// TIA Portal V16 export
// export: Created 2021-09-08T12:46:16.4114193Z, ExportSetting WithDefaults, DisplayName Totally Integrated Automation Portal, DisplayVersion V16 Update 3, DisplayName TIA Portal Version Control Interface, DisplayVersion V16 Update 2, DisplayName TIA Portal Openness, DisplayVersion V16 Update 3, DisplayName TIA Portal Teamcenter Gateway, DisplayVersion V16, DisplayName STEP 7 Professional, DisplayVersion V16 Update 3, DisplayName STEP 7 Safety, DisplayVersion V16, DisplayName WinCC Advanced, DisplayVersion V16 Update 3
TYPE "UF_PARAMETRS"
// stored: IsFailsafeCompliant false
   STRUCT
      Sf : Real;   // Filtration square m2
      flux : Real;
      dP : Real;   // Delta preassure
      Rec : Real;   // Recovery
      Ts : UInt;   // Step time
      Tf : UDInt;   // Filtration time
   END_STRUCT;
END_TYPE
